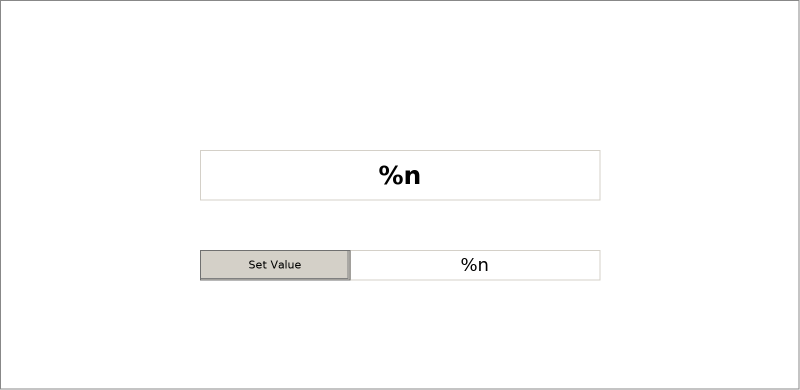
VISUALIZATION VisuKL15XXControl  // 800x390
VAR_IN_OUT
	pDev : POINTER TO FB_DevKL1512;
END_VAR
    Textfield (200,150 400x50), "%n", text variable: pDev^.stManualControl.nCount
    Textfield (350,250 250x30), "%n", text variable: pDev^.stManualControl.nManValue
        OnMouseClick: write the text variable via VisuDialogs.Numpad
    Button (200,250 150x30), "Set Value"
        tap pDev^.stManualControl.bManSetValue
END_VISUALIZATION

(* stored: Version 1.1.0.1, ProductVersion 3.1.4024.11
   Visu VisuKL15XXControl: Id {a31f4940-fba7-09b3-2265-9ff5c4dcceb9} *)
